// TIA Portal V17 export
// export: Created 2023-05-05T14:34:40.4407508Z, ExportSetting None, DisplayName Totally Integrated Automation Portal, DisplayVersion V17, DisplayName TIA Portal Openness, DisplayVersion V17, DisplayName TIA Portal Version Control Interface, DisplayVersion V17, DisplayName SINAMICS Startdrive Advanced, DisplayVersion V17 SP1, DisplayName SINAMICS Startdrive G130, G150, S120, S150, SINAMICS MV, S210, DisplayVersion V17 SP1, DisplayName SINAMICS Startdrive G110M, G120, G120C, G120D, G120P, G115D, DisplayVersion V17 SP1, DisplayName STEP 7 Professional, DisplayVersion V17, DisplayName STEP 7 Safety, DisplayVersion V17, DisplayName WinCC Advanced, DisplayVersion V17
FUNCTION_BLOCK "CompRegulator"   // FB226, FBD
TITLE = CompRegulator / CompFuse
{ S7_Optimized_Access := 'TRUE' }
AUTHOR : XYDNEUBE
FAMILY : N/A
NAME : CompShutter.docx
VERSION : 8.0
// // ===========================================================================
// //
// -----------------------------------------------------------------------------
// // Library:		(that the source is dedicated to)
// // Tested with:	CPU 1516F-3 PN/DP V2.9
// // Engineering:	TIA Portal V17 Update 2
// // Restrictions: 	N/A
// // Requirements: 	N/A
// // Functionality:	Pressure Regulator
// //
// -----------------------------------------------------------------------------
// // Change log table:
// // Version		Date		Expert in charge	Changes applied
// // 00.00.01	12.04.2023	Rahul Kumar	First released version
// //============================================================================
// // ===========================================================================
// //
// -----------------------------------------------------------------------------
// // Library:		(that the source is dedicated to)
// // Tested with:	CPU 1518F-4 V2.6
// // Engineering:	TIA Portal V15 Update 4
// // Restrictions: 	N/A
// // Requirements: 	N/A
// // Functionality:	Fuse
// //
// -----------------------------------------------------------------------------
// // Change log table:
// // Version		Date		Expert in charge	Changes applied
// // 08.00.00	04.03.2020	Dennis Neubert	set rollout to version V8.0
// // 00.00.01	21.11.2018	Dennis Neubert	First released version
// //============================================================================
// stored: IsIECCheckEnabled true, MemoryReserve 100, SetENOAutomatically false
   VAR_IN_OUT
      status : "typeStatusCompRegulator";   // status of component
      status1 : "typeStatusCompRegulator";   // status of component
      configConstant : "typeConfigConstantCompRegulator";   // config constant of component
      hmi : "typeHmiCompRegulator";   // hmi variables to plc and to hmi
   END_VAR
   VAR
      machineInfo { ExternalAccessible := 'False'; ExternalVisible := 'False'; ExternalWritable := 'False'} : "typeMachineInfo";   // Machine information details
      instCompRegulatorError { ExternalAccessible := 'False'; ExternalVisible := 'False'; ExternalWritable := 'False'} : Program_Alarm;   // Componenet Prssure regulator error
      instAlarmCompRegulatorError { ExternalAccessible := 'False'; ExternalVisible := 'False'; ExternalWritable := 'False'} : "PreAlarm";
   END_VAR
   VAR_TEMP
      tempMessageIdError : UDInt;   // message id for Prssure regulator Not valid
      tempMessageNrError : UInt;   // message number Prssure regulatorl Not valid
   END_VAR
   VAR CONSTANT
      STATE_ERROR : UInt := 1;   // message number for Prssure regulator error
   END_VAR
BEGIN

REGION Network 1: ***alarm pressure regulator in Error
   // Error alarms cases are programmed here
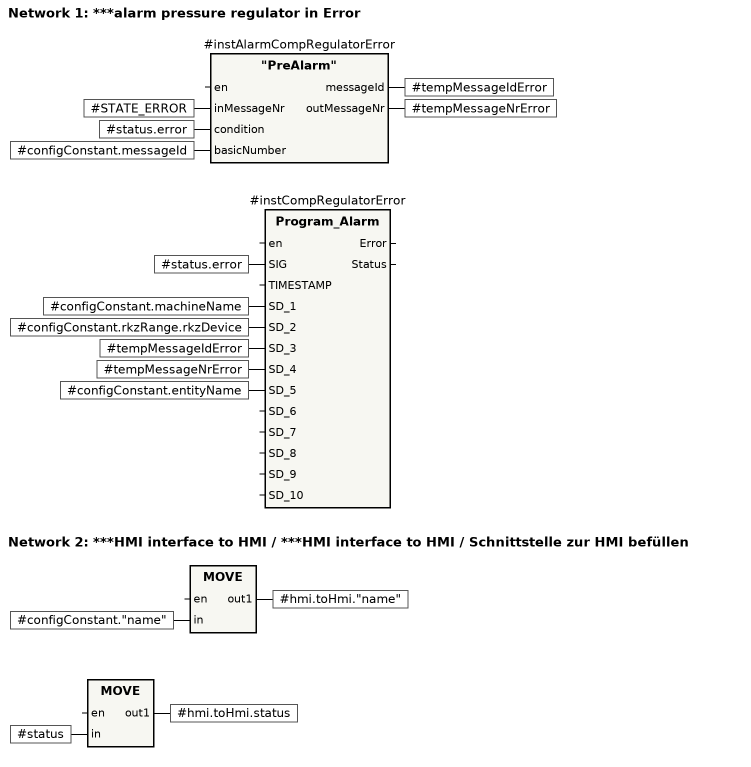
   #instAlarmCompRegulatorError(inMessageNr := #STATE_ERROR,   // "PreAlarm"
                           condition := #status.error,
                           basicNumber := #configConstant.messageId,
                           messageId => #tempMessageIdError,
                           outMessageNr => #tempMessageNrError);
   #instCompRegulatorError(SIG := #status.error,   // Program_Alarm
                           SD_1 := #configConstant.machineName,
                           SD_2 := #configConstant.rkzRange.rkzDevice,
                           SD_3 := #tempMessageIdError,
                           SD_4 := #tempMessageNrError,
                           SD_5 := #configConstant.entityName);
END_REGION

REGION Network 2: ***HMI interface to HMI / ***HMI interface to HMI / Schnittstelle zur HMI befüllen
   // the data which is used by the hmi is transfered to the hmi interface
   #hmi.toHmi."name" := #configConstant."name";
   #hmi.toHmi.status := #status;
END_REGION
END_FUNCTION_BLOCK
